{attribute 'linkalways'} 
{attribute 'no_explicit_call' := 'This FB is a CLASS and must be accessed using methods or properties'}
{attribute 'enable_dynamic_creation'}
FUNCTION_BLOCK _ETcVnAdaptiveThresholdMethod EXTENDS EnumDatatypeBase
VAR
	localData : ETcVnAdaptiveThresholdMethod;
	activeData : REFERENCE TO ETcVnAdaptiveThresholdMethod;
	enumBaseDatatype : _DINT(localData);
END_VAR

METHOD PRIVATE AddLocalEnumeration
VAR_INPUT
	Enumeration : T_MAXSTRING;
	Value : ETcVnAdaptiveThresholdMethod;
END_VAR
AddEnumeration(Enumeration, Value);
END_METHOD

PROPERTY PUBLIC Address : PVOID
GET
Address := ADR(activeData);
END_GET
END_PROPERTY

METHOD PUBLIC ClearReference
VAR_INPUT
END_VAR
activeData REF= localData;
SetBaseDatatypeReference();
END_METHOD

METHOD PUBLIC Clone : I_Datatype
VAR
    pClone : POINTER TO _ETcVnAdaptiveThresholdMethod;
END_VAR
pClone := __NEW(_ETcVnAdaptiveThresholdMethod(InitialValue := Value));
Clone := pClone^;
END_METHOD

METHOD FB_init : BOOL
VAR_INPUT
	bInitRetains : BOOL; // if TRUE, the retain variables are initialized (warm start / cold start)
	bInCopyCode : BOOL;  // if TRUE, the instance afterwards gets moved into the copy code (online change)
	InitialValue : ETcVnAdaptiveThresholdMethod;
END_VAR
localData := InitialValue;
AddBaseDatatype(enumBaseDatatype);
ClearReference();

AddLocalEnumeration('TCVN_ATM_MEAN', ETcVnAdaptiveThresholdMethod.TCVN_ATM_MEAN);
AddLocalEnumeration('TCVN_ATM_GAUSSIAN', ETcVnAdaptiveThresholdMethod.TCVN_ATM_GAUSSIAN);
END_METHOD

PROPERTY PUBLIC Identifier : T_MAXSTRING
GET
Identifier := 'ETcVnAdaptiveThresholdMethod';
END_GET
END_PROPERTY

METHOD IsEnumeratorValueEqual : BOOL
VAR_INPUT
	Enumerator : I_KeyValueForwardEnumerator;
END_VAR
VAR
	storedValue : ETcVnAdaptiveThresholdMethod;
END_VAR
IF NOT Enumerator.TryGet(storedValue) THEN
	RETURN;
END_IF

IsEnumeratorValueEqual := storedValue = activeData;
END_METHOD

METHOD PUBLIC MakeReferenceTo
VAR_INPUT
	ReferenceTarget : REFERENCE TO ETcVnAdaptiveThresholdMethod;
END_VAR
activeData REF= ReferenceTarget;
SetBaseDatatypeReference();
END_METHOD

METHOD PROTECTED SetBaseDatatypeReference
VAR_INPUT
END_VAR
enumBaseDatatype.MakeReferenceTo(activeData);
END_METHOD

PROPERTY PUBLIC Size : UDINT
GET
Size := SIZEOF(activeData);
END_GET
END_PROPERTY

METHOD TryMakeReferenceTo : BOOL
VAR_INPUT
	Target : I_Datatype;
END_VAR
VAR
	targetAsEnum : I_EnumDatatype;
	pTargetData : POINTER TO ETcVnAdaptiveThresholdMethod;
END_VAR
IF NOT Target.TryResolveAsEnumDatatype(targetAsEnum) THEN
	RETURN;
END_IF

IF targetAsEnum.Identifier <> Identifier THEN
	RETURN;
END_IF

pTargetData := Target.Address;
activeData REF= pTargetData^;
SetBaseDatatypeReference();
TryMakeReferenceTo := TRUE;
END_METHOD

PROPERTY PUBLIC Value : ETcVnAdaptiveThresholdMethod
GET
Value := activeData;
END_GET
SET
activeData := Value;
END_SET
END_PROPERTY

END_FUNCTION_BLOCK

(* stored: Version 1.1.0.1, ProductVersion 3.1.4024.12
   POU _ETcVnAdaptiveThresholdMethod: Id {07ab21eb-1ccb-0124-2480-afbf70a289da}, SpecialFunc None
   Folder Constructor: Id {e0ffc21e-78a3-03bd-3bc2-022c66c6b4c8}
   Folder Private: Id {f6c770e6-12a8-0a04-33a2-130ed4c74e3d}
   Folder Protected: Id {97d0bb06-317b-03a0-2e8a-4f761dae8ef9}
   Method AddLocalEnumeration: Id {a6a8d712-19f2-0ae3-2f36-361c62c2f67a}
   Property Address: Id {e73b6060-fa4d-010a-143f-0b96a620cf32}
   Get Get: Id {693c20d4-f86a-0d2c-0583-bb3c677deb53}
   Method ClearReference: Id {01d22aea-e07e-0f30-080b-71e320a7be50}
   Method Clone: Id {b404cb6b-a483-027d-2b87-2a1e4e56179a}
   Method FB_init: Id {ce50a230-b848-0bdd-06e0-90bf5d7fe54a}
   Property Identifier: Id {c369b410-307b-05c6-3c61-41183f8284ed}
   Get Get: Id {6798af16-ac2c-0887-3646-b36d8def19a0}
   Method IsEnumeratorValueEqual: Id {cbf4504d-d37a-0556-3553-d617343e2915}
   Method MakeReferenceTo: Id {ae3895c6-9fac-02bd-04a5-33a381f66f4b}
   Method SetBaseDatatypeReference: Id {573c46b0-b1ca-0a29-3ad4-20eaf4bfc27d}
   Property Size: Id {43152bfc-b67d-0644-3b73-7229e83fc928}
   Get Get: Id {790f9e5c-18b9-0d10-398a-5746dc25111b}
   Method TryMakeReferenceTo: Id {48af6bec-7e8b-036d-16c8-b74683f99161}
   Property Value: Id {1dc71022-d7c2-062f-11a6-e51e05afa909}
   Get Get: Id {9ac64dc2-b906-0f7b-3619-169929997308}
   Set Set: Id {cc723d01-6e00-07a2-2954-975cc28bf7f8} *)
